// struct for sending data to 
TYPE ARCommunicationSendPacket_t :
STRUCT
	
END_STRUCT
END_TYPE

(* stored: Version 1.1.0.1
   DUT ARCommunicationSendPacket_t: Id {1496e6dd-61d0-4dc4-9fe0-fce58ff7662a} *)
